TYPE
  (* Standard: 61499-1 *)
  (* Version 1.0, 2026-05-26, Dimitrios Kalligaridis *)
  PACKAGE mypackage;
  OuterStruct : STRUCT
    inner : mypackage::InnerStruct;
  END_STRUCT;
END_TYPE
